{attribute 'hide_all_locals'}
FUNCTION_BLOCK FB_LinkedList_Node IMPLEMENTS ITF_LinkedList_Node

VAR
	itf_ListNext:		ITF_LinkedList_Node;
	itf_ListPrevious:	ITF_LinkedList_Node;
	itf_LinkMaster:		ITF_LinkedList_Master;
	
	{attribute 'no_copy'}
	_bInCopyCode : 		BOOL;
END_VAR

METHOD FB_exit : BOOL
VAR_INPUT
	bInCopyCode : BOOL; // if TRUE, the exit method is called for exiting an instance that is copied afterwards (online change).
END_VAR
IF NOT bInCopyCode THEN
	//Destroy and remove from list
	IF itf_LinkMaster <> 0 THEN
		itf_LinkMaster.mListRemove( THIS^ );
	END_IF
END_IF
END_METHOD

METHOD FB_init : BOOL
VAR_INPUT
	bInitRetains : 	BOOL; // if TRUE, the retain variables are initialized (warm start / cold start)
	bInCopyCode : 	BOOL;  // if TRUE, the instance afterwards gets moved into the copy code (online change)
END_VAR
_bInCopyCode 	:= bInCopyCode;
END_METHOD

METHOD FB_reinit : BOOL
VAR_INPUT
END_VAR
_bInCopyCode := FALSE; //Next set of p_LinkMaster wont be from initializing new instance during copy
END_METHOD

PROPERTY p_IsLinkMaster : BOOL
GET
p_IsLinkMaster := FALSE;
END_GET
END_PROPERTY

PROPERTY p_LinkMaster : ITF_LinkedList_Master
GET
p_LinkMaster := itf_LinkMaster;
END_GET
SET
IF NOT _bInCopyCode THEN //Set not called during process of copying function block
	
	IF itf_LinkMaster <> 0 THEN
		//Remove from old master
		itf_LinkMaster.mListRemove( THIS^ );
	END_IF

	IF p_LinkMaster <> 0 THEN
		//Add to new master
		p_LinkMaster.mListAdd( THIS^ );
		//Store master
		itf_LinkMaster := p_LinkMaster;
	END_IF

END_IF
END_SET
END_PROPERTY

PROPERTY p_ListNext : ITF_LinkedList_Node
GET
p_ListNext := itf_ListNext;
END_GET
SET
itf_ListNext := p_ListNext;
END_SET
END_PROPERTY

PROPERTY p_ListPrevious : ITF_LinkedList_Node
GET
p_ListPrevious := itf_ListPrevious;
END_GET
SET
itf_ListPrevious := p_ListPrevious;
END_SET
END_PROPERTY

END_FUNCTION_BLOCK

(* stored: Version 1.1.0.1, ProductVersion 3.1.4024.12
   POU FB_LinkedList_Node: Id {90324853-2e5f-49f8-8220-eae435ca271f}, SpecialFunc None
   Method FB_exit: Id {fa2242ef-60a6-0868-3bec-653fb43dd7fb}
   Method FB_init: Id {b0701d5a-3a14-05ed-381a-206b7903b86d}
   Method FB_reinit: Id {4813a597-044b-43a1-991e-2307a175fc43}
   Property p_IsLinkMaster: Id {17f08b8b-3c60-4702-bfc6-070a986dfc0c}
   Get Get: Id {0990a748-3c52-4160-af65-bc1a7d44b7c0}
   Property p_LinkMaster: Id {6076d27c-543e-491b-82fc-59b02048ee72}
   Get Get: Id {51931b2a-3baa-4776-ad59-fab0b175695c}
   Set Set: Id {1c3e8a69-b5ff-44dd-9260-37ec38464d00}
   Property p_ListNext: Id {f41588f3-e43c-4372-8a12-18f9caf92429}
   Get Get: Id {4ade9195-19e2-4299-acdf-9880f7faef05}
   Set Set: Id {67f5a8b1-870d-4fb1-a4c9-6e8c5f1e5aaa}
   Property p_ListPrevious: Id {21cc6a69-d3da-400d-81b9-854f8aa2122d}
   Get Get: Id {a9c21024-3b02-43d7-bc3f-b1ac2bb904e8}
   Set Set: Id {755fe7ff-a81c-42c8-8e0a-126358d187bb} *)
